Fanuc KAREL source: SUB_STR.kl

PROGRAM T
%NOLOCKGROUP
VAR
 v0 : STRING[40]
 v1 : INTEGER
 v2 : INTEGER
 res : STRING[40]
BEGIN
 res = SUB_STR(v0, v1, v2)
END T
